{attribute 'TcGenerated'}
{attribute 'no-analysis'}
{attribute 'linkalways'}
// This function has been automatically generated from the project information.
VAR_GLOBAL CONSTANT
	{attribute 'const_non_replaced'}
	stLibVersion_Tk_SystemControl : ST_LibVersion := (iMajor := 0, iMinor := 0, iBuild := 5, iRevision := 0, nFlags := 0, sVersion := '0.0.5.0');
END_VAR

(* stored: Version 1.1.0.1
   GVL Global_Version: Id {45c9a5c3-4008-47c5-9768-8f277b5e76a2} *)
